FUNCTION HOUR_TO_DEG : LREAL
VAR_INPUT
    hours : LREAL;
END_VAR
VAR
END_VAR

HOUR_TO_DEG := hours / 24.0 * 360.0;

END_FUNCTION

(* stored: Version 1.1.0.1, ProductVersion 3.1.4019.2
   POU HOUR_TO_DEG: Id {f0500d32-5a74-4de0-b74c-06ec2f5d27c2}, SpecialFunc None *)
